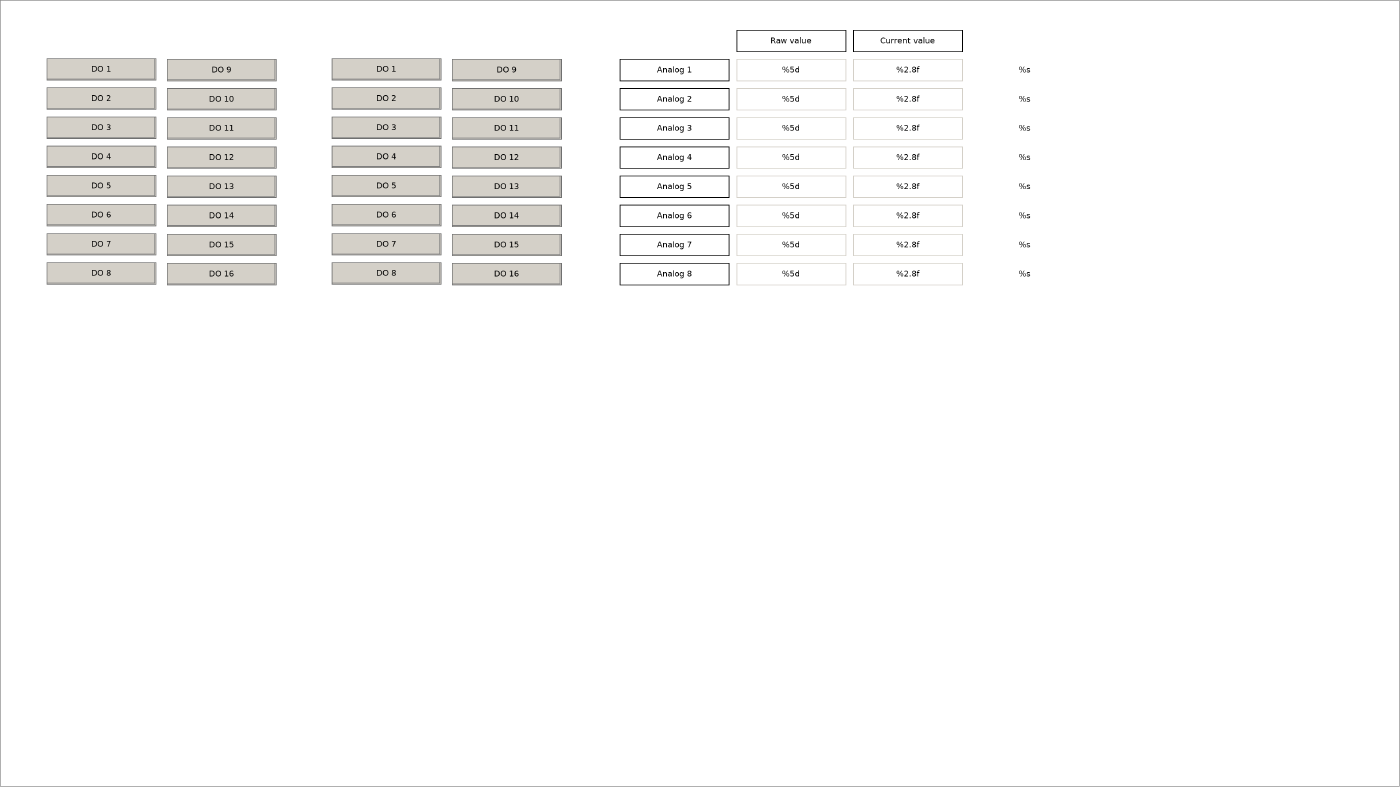
VISUALIZATION Visualization  // 1920x1080
    Button (64,80 150x30), "DO 1", colour toggle: MAIN.bDO11
        toggle MAIN.bDO11
    Button (64,120 150x30), "DO 2", colour toggle: MAIN.bDO12
        toggle MAIN.bDO12
    Button (64,160 150x30), "DO 3", colour toggle: MAIN.bDO13
        toggle MAIN.bDO13
    Button (64,200 150x30), "DO 4", colour toggle: MAIN.bDO14
        toggle MAIN.bDO14
    Button (64,240 150x30), "DO 5", colour toggle: MAIN.bDO15
        toggle MAIN.bDO15
    Button (64,280 150x30), "DO 6", colour toggle: MAIN.bDO16
        toggle MAIN.bDO16
    Button (64,320 150x30), "DO 7", colour toggle: MAIN.bDO17
        toggle MAIN.bDO17
    Button (64,360 150x30), "DO 8", colour toggle: MAIN.bDO18
        toggle MAIN.bDO18
    Button (229,81 150x30), "DO 9", colour toggle: MAIN.bDO19
        toggle MAIN.bDO19
    Button (229,121 150x30), "DO 10", colour toggle: MAIN.bDO110
        toggle MAIN.bDO110
    Button (229,161 150x30), "DO 11", colour toggle: MAIN.bDO111
        toggle MAIN.bDO111
    Button (229,201 150x30), "DO 12", colour toggle: MAIN.bDO112
        toggle MAIN.bDO112
    Button (229,241 150x30), "DO 13", colour toggle: MAIN.bDO113
        toggle MAIN.bDO113
    Button (229,281 150x30), "DO 14", colour toggle: MAIN.bDO114
        toggle MAIN.bDO114
    Button (229,321 150x30), "DO 15", colour toggle: MAIN.bDO115
        toggle MAIN.bDO115
    Button (229,361 150x30), "DO 16", colour toggle: MAIN.bDO116
        toggle MAIN.bDO116
    Button (455,80 150x30), "DO 1", colour toggle: MAIN.bDO21
        toggle MAIN.bDO21
    Button (455,120 150x30), "DO 2", colour toggle: MAIN.bDO22
        toggle MAIN.bDO22
    Button (455,160 150x30), "DO 3", colour toggle: MAIN.bDO23
        toggle MAIN.bDO23
    Button (455,200 150x30), "DO 4", colour toggle: MAIN.bDO24
        toggle MAIN.bDO24
    Button (455,240 150x30), "DO 5", colour toggle: MAIN.bDO25
        toggle MAIN.bDO25
    Button (455,280 150x30), "DO 6", colour toggle: MAIN.bDO26
        toggle MAIN.bDO26
    Button (455,320 150x30), "DO 7", colour toggle: MAIN.bDO27
        toggle MAIN.bDO27
    Button (455,360 150x30), "DO 8", colour toggle: MAIN.bDO28
        toggle MAIN.bDO28
    Button (620,81 150x30), "DO 9", colour toggle: MAIN.bDO29
        toggle MAIN.bDO29
    Button (620,121 150x30), "DO 10", colour toggle: MAIN.bDO210
        toggle MAIN.bDO210
    Button (620,161 150x30), "DO 11", colour toggle: MAIN.bDO211
        toggle MAIN.bDO211
    Button (620,201 150x30), "DO 12", colour toggle: MAIN.bDO212
        toggle MAIN.bDO212
    Button (620,241 150x30), "DO 13", colour toggle: MAIN.bDO213
        toggle MAIN.bDO213
    Button (620,281 150x30), "DO 14", colour toggle: MAIN.bDO214
        toggle MAIN.bDO214
    Button (620,321 150x30), "DO 15", colour toggle: MAIN.bDO215
        toggle MAIN.bDO215
    Button (620,361 150x30), "DO 16", colour toggle: MAIN.bDO216
        toggle MAIN.bDO216
    Rectangle (850,81 150x30), "Analog 1"
    Rectangle (850,121 150x30), "Analog 2"
    Rectangle (850,201 150x30), "Analog 4"
    Rectangle (850,161 150x30), "Analog 3"
    Rectangle (850,281 150x30), "Analog 6"
    Rectangle (850,241 150x30), "Analog 5"
    Rectangle (850,321 150x30), "Analog 7"
    Rectangle (850,361 150x30), "Analog 8"
    Textfield (1170,81 150x30), "%2.8f", text variable: MAIN.lrGovernorGuideVaneOilPreesure
    Textfield (1170,121 150x30), "%2.8f", text variable: MAIN.lrGovernorBladeOilPressure
    Textfield (1170,161 150x30), "%2.8f", text variable: MAIN.lrExcitationVoltage
    Textfield (1170,201 150x30), "%2.8f", text variable: MAIN.lrExcitationCurrent
    Textfield (1170,241 150x30), "%2.8f", text variable: MAIN.lrSpiralCasePressure
    Textfield (1170,281 150x30), "%2.8f", text variable: MAIN.lrHeadCasePressure
    Textfield (1170,321 150x30), "%2.8f", text variable: MAIN.lrDraftT1CasePressure
    Textfield (1170,361 150x30), "%2.8f", text variable: MAIN.lrDraftT2CasePressure
    Rectangle (1170,41 150x30), "Current value"
    Rectangle (1330,81 150x30), "%s", text variable: MAIN.fbCal1.sDescription
    Rectangle (1330,121 150x30), "%s", text variable: MAIN.fbCal2.sDescription
    Rectangle (1330,201 150x30), "%s", text variable: MAIN.fbCal4.sDescription
    Rectangle (1330,161 150x30), "%s", text variable: MAIN.fbCal3.sDescription
    Rectangle (1330,281 150x30), "%s", text variable: MAIN.fbCal6.sDescription
    Rectangle (1330,241 150x30), "%s", text variable: MAIN.fbCal5.sDescription
    Rectangle (1330,321 150x30), "%s", text variable: MAIN.fbCal7.sDescription
    Rectangle (1330,361 150x30), "%s", text variable: MAIN.fbCal8.sDescription
    Textfield (1010,81 150x30), "%5d", text variable: MAIN.fbCal1.wRawIn
    Textfield (1010,121 150x30), "%5d", text variable: MAIN.fbCal2.wRawIn
    Textfield (1010,161 150x30), "%5d", text variable: MAIN.fbCal3.wRawIn
    Textfield (1010,201 150x30), "%5d", text variable: MAIN.fbCal4.wRawIn
    Textfield (1010,241 150x30), "%5d", text variable: MAIN.fbCal5.wRawIn
    Textfield (1010,281 150x30), "%5d", text variable: MAIN.fbCal6.wRawIn
    Textfield (1010,321 150x30), "%5d", text variable: MAIN.fbCal7.wRawIn
    Textfield (1010,361 150x30), "%5d", text variable: MAIN.fbCal8.wRawIn
    Rectangle (1010,41 150x30), "Raw value"
END_VISUALIZATION

(* stored: Version 1.1.0.1, ProductVersion 3.1.4024.11
   Visu Visualization: Id {7cd2cbed-36c9-41c1-b386-6080408a2b81} *)
